FUNCTION_BLOCK AX_FB_TOF_LTIME (* standard timer function block (off-delay timing) with AX Adapter *)
  (* Standard: 61131-3; Classification: standard timer function block; Description: Copyright (c) 2011 TU Wien ACIN, HR Agrartechnik GmbH This program and the accompanying materials are made available under the terms of the Eclipse Public License 2.0 which is available at https://www.eclipse.org/legal/epl-2.0/ SPDX-License-Identifier: EPL-2.0 *)
  (* Version 3.0, 2025-04-14, Patrick Aigner, changed package *)
  (* Version 1.0, 2011-06-21, Monika Wenger, TU Wien ACIN, initial API and implementation and/or initial documentation *)
  PACKAGE adapter::iec61131::timers;
  IMPORT eclipse4diac::core::TypeHash;
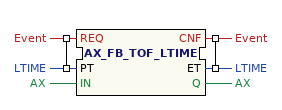
  EVENT_INPUT
    REQ WITH PT; (* Normal Execution Request (non-triggering) *)
  END_EVENT
  EVENT_OUTPUT
    CNF WITH ET; (* Execution Confirmation *)
  END_EVENT
  VAR_INPUT
    PT : LTIME; (* Process time *)
  END_VAR
  VAR_OUTPUT
    ET : LTIME; (* Elapsed time *)
  END_VAR
  SOCKETS
    IN : adapter::types::unidirectional::AX; (* Input *)
  END_SOCKETS
  PLUGS
    Q : adapter::types::unidirectional::AX; (* Output *)
  END_PLUGS
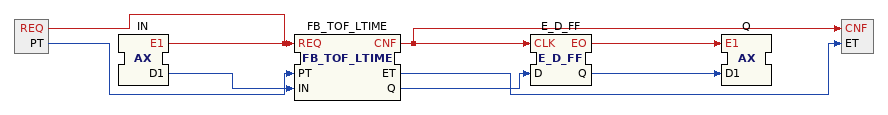
  FBS
    FB_TOF_LTIME : iec61131::timers::FB_TOF_LTIME;
    E_D_FF : iec61499::events::E_D_FF;
  END_FBS
  EVENT_CONNECTIONS
    IN.E1 TO FB_TOF_LTIME.REQ;
    FB_TOF_LTIME.CNF TO E_D_FF.CLK;
    E_D_FF.EO TO Q.E1;
    REQ TO FB_TOF_LTIME.REQ;
    FB_TOF_LTIME.CNF TO CNF;
  END_CONNECTIONS
  DATA_CONNECTIONS
    FB_TOF_LTIME.ET TO ET;
    PT TO FB_TOF_LTIME.PT;
    IN.D1 TO FB_TOF_LTIME.IN;
    FB_TOF_LTIME.Q TO E_D_FF.D;
    E_D_FF.Q TO Q.D1;
  END_CONNECTIONS
END_FUNCTION_BLOCK
